// TIA Portal V20 export
VAR_GLOBAL   // PLC tag table "Inputs Machine"
END_VAR
